Staubli VAL3: Deb2403.pjx

--- Deb2403.pjx ---
Parameters version=s7.4 stackSize=5000 millimeterUnit=true
Program file=main.pgx
Program file=prgm1.pgx
Program file=start.pgx
Program file=stop.pgx
Data file=Deb2403.dtx

--- Deb2403.dtx ---
mdesc mNomSpeed = {accel=200, vel=400, decel=200}
dio EntreePwrl0 = {link=POWERLINK-1\%I0}
dio SortiePwrl0 = {link=POWERLINK-1\%Q0}
tool tTool = {z=67, fatherId=flange[0], ioLink=valve1}
jointRx jP1
jointRx jP2 = {j1=67.72, j2=50.87, j3=100.24, j5=28.89, j6=-112.28}
jointRx jP3 = {j1=-83.94, j2=66.93, j3=62.59, j5=50.48, j6=-263.94}
jointRx jP4 = {j1=67.72, j2=17.89, j3=90, j5=72.11, j6=-112.28}
jointRx jP5 = {j1=-84.94, j2=43.97, j3=50.35, j5=58.68, j6=-263.94}
frame fFrame = {x=-421.67, y=-92.07, z=-232.31, rx=0.62, ry=178.2, rz=-83.18, fatherId=world[0]}

--- main.pgx ---
program main()
begin
  while true
    doECAT1_0 = true

    if(diECAT1_0 == true)

      doECAT1_0 = false

      x[0] = diECAT1_1
      x[1] = diECAT1_2
      x[2] = diECAT1_3
      x[3] = diECAT1_4
      x[4] = diECAT1_5
      x[5] = diECAT1_6
      x[6] = diECAT1_7
      x[7] = diECAT1_8

      co_x = x[0] * 1 + x[1] * 2 + x[2] * 4 + x[3] * 8 + x[4] * 16 + x[5] * 32 + x[6] * 64 + x[7] * 128

      y[0] = diECAT1_9
      y[1] = diECAT1_10
      y[2] = diECAT1_11
      y[3] = diECAT1_12
      y[4] = diECAT1_13
      y[5] = diECAT1_14
      y[6] = diECAT1_15
      y[7] = diECAT1_16

      co_y = y[0] * 1 + y[1] * 2 + y[2] * 4 + y[3] * 8 + y[4] * 16 + y[5] * 32 + y[6] * 64 + y[7] * 128

      open(tTool)
      movej(jP1, tTool, mNomSpeed)
      movej(jP2, tTool, mNomSpeed)
      close(tTool)
      movej(jP4, tTool, mNomSpeed)
      movej(jP5, tTool, mNomSpeed)
      movej(jP3, tTool, mNomSpeed)
      open(tTool)
      movej(jP1, tTool, mNomSpeed)
      movej(jP3, tTool, mNomSpeed)
      close(tTool)
      movej(jP5, tTool, mNomSpeed)
      movej(jP4, tTool, mNomSpeed)
      movej(jP2, tTool, mNomSpeed)
      open(tTool)

      doECAT1_0 = true

    endIf
  endWhile
end

--- start.pgx ---
program start()
begin
      call prgm1()
end

--- prgm1.pgx ---
program prgm1()
begin
  while true
    if(EntreePwrl0==true)
      open(tTool)
      movej(jP1, tTool, mNomSpeed)
      movej(jP2, tTool, mNomSpeed)
      close(tTool)
      movej(jP4, tTool, mNomSpeed)
      movej(jP5, tTool, mNomSpeed)
      movej(jP3, tTool, mNomSpeed)
      open(tTool)
      movej(jP1, tTool, mNomSpeed)
      movej(jP3, tTool, mNomSpeed)
      close(tTool)
      movej(jP5, tTool, mNomSpeed)
      movej(jP4, tTool, mNomSpeed)
      movej(jP2, tTool, mNomSpeed)
      open(tTool)
      waitEndMove()
    endIf
  endWhile
end

--- test_com.pgx ---
program test_com()
begin
  while true
    doECAT1_0 = true

    if(diECAT1_0 == true)

      doECAT1_0 = false

      open(tTool)
      movej(jP1, tTool, mNomSpeed)
      movej(jP2, tTool, mNomSpeed)
      close(tTool)
      movej(jP4, tTool, mNomSpeed)
      movej(jP5, tTool, mNomSpeed)
      movej(jP3, tTool, mNomSpeed)
      open(tTool)
      movej(jP1, tTool, mNomSpeed)
      movej(jP3, tTool, mNomSpeed)
      close(tTool)
      movej(jP5, tTool, mNomSpeed)
      movej(jP4, tTool, mNomSpeed)
      movej(jP2, tTool, mNomSpeed)
      open(tTool)
      waitEndMove()

      doECAT1_0 = true

    endIf
  endWhile
end
